# EPICS substitutions: ek9000App/Db/EL3078.substitutions
file EL3078.template
{       pattern
        {
                TERMINAL,

        }
        {
        }
}
